PROGRAM Step_2_StickMachine // Stick Machine
VAR
	
	// Internals 
	JOGStickConveyorFWD : BOOL;     // set from HMI
	JOGStickFeedChainFWD : BOOL;   // set from HMI
	LocalSafety_2: BOOL;             //Safety Conditions
	
	
	 // Edge detectors
    rtStart : R_TRIG;      // Rising edge Cycle Start
    rtStop  : R_TRIG;      // Rising edge Cycle Stop
	
	
	
	// Timers 
    tHoistPause  : TON;         // Running time for Stick conveyor and feed chain after tilt hoist reaches bottom limit switch
	
	
	
END_VAR

// Safety
LocalSafety_2 := StickConveyorMMP AND StickFeedChainMMP;



// Defaults: make outputs known each scan
Step2_RedFlash    := FALSE;
Step2_RedSteady    := FALSE;
Step2_YellowSteady := FALSE;
Step2_YellowFlash := FALSE;
Step2_GreenSteady  := FALSE;
Step2_GreenFlash  := FALSE;
StickConveyorFWD := FALSE;
StickFeedChainFWD := FALSE;


// Edge detect PBs and Optical falling edge
rtStart(CLK := CycleStartPB);
rtStop(CLK := CycleStopPB);


// Stop button or lost permissive or lost local safety → go to IDLE immediately
IF (rtStop.Q OR NOT Permissive OR NOT LocalSafety_2) THEN
    Step2_State := 0;        // IDLE
END_IF;




// -------------------- Manual override (when AutoMode = FALSE) ------------------
IF NOT AutoMode THEN
    // Simple, safe manual jogs
    IF JOGStickConveyorFWD  AND Permissive AND LocalSafety_2 THEN
        StickConveyorFWD := TRUE;
	ELSE
		StickConveyorFWD := FALSE;
    END_IF

    IF JOGStickFeedChainFWD AND Permissive AND LocalSafety_2 THEN
        StickFeedChainFWD := TRUE;
	ELSE
		StickFeedChainFWD := FALSE;
    END_IF

    // Tower lights in manual: Yellow
    IF NOT AutoMode THEN
        Step2_YellowSteady := TRUE;
    END_IF

    RETURN;    // skips Auto sequence when in manual
END_IF



    // ---------------------- Auto Sequence-------------------------------------

CASE Step2_State OF

    0:  // IDLE / READY
        Step2_YellowSteady := TRUE;
        StickConveyorFWD   := FALSE;
        StickFeedChainFWD  := FALSE;

        // If safe and not full, wait for Step 1 pause or start signal
        IF (Permissive AND LocalSafety_2 AND NOT StickMachine_TopLimit) THEN
            IF rtStart.Q THEN
                Step2_State := 10;      // start feeding
            END_IF
        END_IF


    // ---------------------------------------------------
    10: // RUNNING / FEEDING
     
		Step2_RedFlash    := FALSE;
		Step2_RedSteady    := FALSE;
		Step2_YellowSteady := FALSE;
		Step2_YellowFlash := FALSE;
		Step2_GreenSteady  := TRUE;
		Step2_GreenFlash  := FALSE;
        StickConveyorFWD  := TRUE;
        StickFeedChainFWD := TRUE;
		
		UnscramblerDelay(IN := UnscramblerBoardDetected, PT := T#30S);	
		 tHoistPause(IN := Step1_YellowFlash OR UnscramblerDelay.IN, PT := T#30S); // Tilt hoist reaches bottom limit and timer start, stickmachine motors run for set time after tilt hoist reaches bottom
		
        // Stop when bin becomes full or Tilt Hoist is at bottom
        IF StickMachine_TopLimit OR tHoistPause.Q (*OR Step2OffSignal*)THEN
            StickConveyorFWD  := FALSE;
            StickFeedChainFWD := FALSE;
			StopStep3 := TRUE;
            Step2_State := 20;          // go to FULL / FLASH
        END_IF

        // Lost safety or permissive → back to IDLE
        IF (NOT Permissive) OR (NOT LocalSafety_2) THEN
            StickConveyorFWD  := FALSE;
            StickFeedChainFWD := FALSE;
            Step2_State := 0;
        END_IF


    // ---------------------------------------------------
    20: // FULL BIN / Yellow FLASH
        Step2_RedFlash    := FALSE;
		Step2_RedSteady    := FALSE;
		Step2_YellowSteady := FALSE;
		Step2_YellowFlash := TRUE;
		Step2_GreenSteady  := FALSE;
		Step2_GreenFlash  := FALSE;
        StickConveyorFWD   := FALSE;
        StickFeedChainFWD  := FALSE;
		
       
        IF rtStart.Q AND NOT StickMachine_TopLimit AND Permissive AND LocalSafety_2 THEN
			Step2_YellowFlash := FALSE;
            Step2_State := 10;          // go to running
        END_IF


END_CASE

END_PROGRAM

(* stored: Version 1.1.0.1
   POU Step_2_StickMachine: Id {b4dc1e3c-4140-4c36-bc6c-90124021e85e}, SpecialFunc None *)
